TYPE ST_Control :
STRUCT
	ClearAllFault : BOOL;
	Abort		  : BOOL;
END_STRUCT
END_TYPE

(* stored: Version 1.1.0.1, ProductVersion 3.1.4024.11
   DUT ST_Control: Id {dfe63870-8943-4f6e-a0e1-1654f728e76d} *)
